FUNCTION_BLOCK IntPointerComparer EXTENDS Object IMPLEMENTS IPointerComparer
VAR
	_ClassName : STRING := __POUNAME();
END_VAR

{attribute 'monitoring' := 'call'}
PROPERTY ClassName : STRING
GET
ClassName := _ClassName;
END_GET
END_PROPERTY

{attribute "object_name" := "Compare"}
METHOD Compare : COMPARISION_RESULT
VAR_INPUT
	left : PVOID;
	right : PVOID;
END_VAR
VAR
	leftPointer : POINTER TO INT; 
	rightPointer : POINTER TO INT; 
END_VAR
IF left = 0 AND right = 0 THEN
	Compare := COMPARISION_RESULT.FIRST_EQUAL_TO_SECOND;
	RETURN;
END_IF

IF left = 0 THEN
	Compare := COMPARISION_RESULT.FIRST_LESS_THAN_SECOND;
	RETURN;	
END_IF

IF right = 0 THEN
	Compare := COMPARISION_RESULT.FIRST_GREATER_THAN_SECOND;
	RETURN;	
END_IF

leftPointer := left;
rightPointer := right;

IF leftPointer^ < rightPointer^ THEN
	Compare := COMPARISION_RESULT.FIRST_LESS_THAN_SECOND;
ELSIF leftPointer^ > rightPointer^ THEN
	Compare := COMPARISION_RESULT.FIRST_GREATER_THAN_SECOND;
ELSE
	Compare := COMPARISION_RESULT.FIRST_EQUAL_TO_SECOND;	
END_IF
END_METHOD

{attribute 'monitoring' := 'call'}
PROPERTY Size : ULINT
GET
Size := XSIZEOF(THIS^);
END_GET
END_PROPERTY

END_FUNCTION_BLOCK

(* stored: Version 1.1.0.1
   POU IntPointerComparer: Id {2c0225a9-2344-4d20-814a-704440543b13}, SpecialFunc None
   Property ClassName: Id {a7cff5f3-499b-4842-989e-2bb2df27d245}
   Get Get: Id {f12116d1-e140-4a1f-8a25-fc9f6616739d}
   Method Compare: Id {c4ce0496-02a1-4d62-8be5-2c807767f44a}
   Property Size: Id {6e076afb-34bc-4a65-979c-cc966b3b7e37}
   Get Get: Id {85ba2351-dd71-4a0f-bcc9-2352180520e5} *)
